{attribute 'qualified_only'}
VAR_GLOBAL
	Black	: TcVnVector4_LREAL := [0,0,0,0];
	White	: TcVnVector4_LREAL := [255,255,255,0];

	Maroon	: TcVnVector4_LREAL := [128,0,0,0];
	Red		: TcVnVector4_LREAL := [255,0,0,0];
	Orange	: TcVnVector4_LREAL := [255,165,0,0];
	Yellow	: TcVnVector4_LREAL := [255,255,0,0];
	Olive	: TcVnVector4_LREAL := [128,128,0,0];
	Green	: TcVnVector4_LREAL := [0,128,0,0];
	Purple	: TcVnVector4_LREAL := [128,0,128,0];
	Fuchsia	: TcVnVector4_LREAL := [255,0,255,0];
	Lime	: TcVnVector4_LREAL := [0,255,0,0];
	Teal	: TcVnVector4_LREAL := [0,128,128,0];
	Aqua	: TcVnVector4_LREAL := [0,255,255,0];
	Blue	: TcVnVector4_LREAL := [0,0,255,0];
	Navy	: TcVnVector4_LREAL := [0,0,128,0];
	Gray	: TcVnVector4_LREAL := [128,128,128,0];
	Silver	: TcVnVector4_LREAL := [192,192,192,0];

END_VAR

(* stored: Version 1.1.0.1
   GVL Color: Id {e4a178e0-704b-45ee-bae1-b18eebbd48de} *)
